(*
SPDX-FileCopyrightText: © 2026 Oleksandr Tiutyk <trofimich@gmail.com>
SPDX-License-Identifier: MIT
License: https://opensource.org/license/mit
*)

(*!
<summary>
Beckhoff EL3078: 8-channel multi-range analog input terminal (REAL values).
</summary>
<description>
Process image mapping structure for the EL3078 EtherCAT terminal with 8 multi-range analog input channels
outputting REAL floating-point values.
Requires AI Standard (Real32) TxPDOs 0x1A10, 0x1A12, 0x1A14, 0x1A16, 0x1A18, 0x1A1A, 0x1A1C and 0x1A1E.
Value entries at 0x60n0:13 are REAL32; INT16 and compact assignments are outside this model.
When used for I/O, link located fields or their containing buffers to the matching selected PDOs.
The record is not a packed wire buffer; compiler padding is not part of the device specification.
Unlinked/default values do not prove valid I/O. The caller evaluates bus/channel validity before use.
Use one owner task per instance and externally synchronize other access; multi-field snapshots are not atomic.
Copies store data without creating hardware links. Keep borrowed field references valid while consumers are bound.
This passive record performs no validation, synchronization, configuration or protocol advancement.
Select standard status-plus-value PDOs matching the declared Value type; compact value-only PDOs
are outside this model. Configure electrical range and scaling separately on the device.
</description>
*)
TYPE EL3078 :
STRUCT
	Ch1 : ANALOG_INPUT_REAL_CHANNEL;
	Ch2 : ANALOG_INPUT_REAL_CHANNEL;
	Ch3 : ANALOG_INPUT_REAL_CHANNEL;
	Ch4 : ANALOG_INPUT_REAL_CHANNEL;
	Ch5 : ANALOG_INPUT_REAL_CHANNEL;
	Ch6 : ANALOG_INPUT_REAL_CHANNEL;
	Ch7 : ANALOG_INPUT_REAL_CHANNEL;
	Ch8 : ANALOG_INPUT_REAL_CHANNEL;
END_STRUCT
END_TYPE

(* stored: Version 1.1.0.1, ProductVersion 3.1.4026.20
   DUT EL3078: Id {c6b3c33b-6858-4075-bee5-bd3047b70644} *)
